SUBAPPLICATION Granulatschieber (* Subapplication Type *)
  (* Standard: 61499-2 *)
  (* Version 1.0, 2024-04-23, Elias *)
  IMPORT DataPanel::io::MI::DQ::DataPanel_MI_DO::DigitalOutput_1A;
  IMPORT DataPanel::io::MI::const::MI::MI_00;
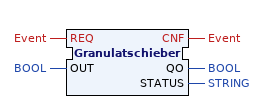
  EVENT_INPUT
    REQ;
  END_EVENT
  EVENT_OUTPUT
    CNF;
  END_EVENT
  VAR_INPUT
    OUT : BOOL;
  END_VAR
  VAR_OUTPUT
    QO : BOOL;
    STATUS : STRING;
  END_VAR
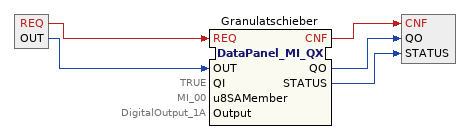
  FBS
    Granulatschieber : DataPanel::io::MI::DQ::DataPanel_MI_QX(QI := TRUE, u8SAMember := MI_00, Output := DigitalOutput_1A);
  END_FBS
  EVENT_CONNECTIONS
    REQ TO Granulatschieber.REQ;
    Granulatschieber.CNF TO CNF;
  END_CONNECTIONS
  DATA_CONNECTIONS
    OUT TO Granulatschieber.OUT;
    Granulatschieber.QO TO QO;
    Granulatschieber.STATUS TO STATUS;
  END_CONNECTIONS
END_SUBAPPLICATION
